KUKA KRL program: chk_w7_grp1_vac.src

&ACCESS RVO10
&COMMENT vacuo GRP axor
DEF chk_w7_grp1_vac( )

; Check Vacuum on gripper AXOR
;//---- Start User-------

$TIMER[10] = 0
$TIMER_STOP[10] = FALSE

WAIT FOR ($IN[493])

$TIMER_STOP[10] = TRUE
$TIMER[10] = 0

;//---- End User---------
END
